Universal Robots PolyScope program: stopCollarMoveBottle.urp

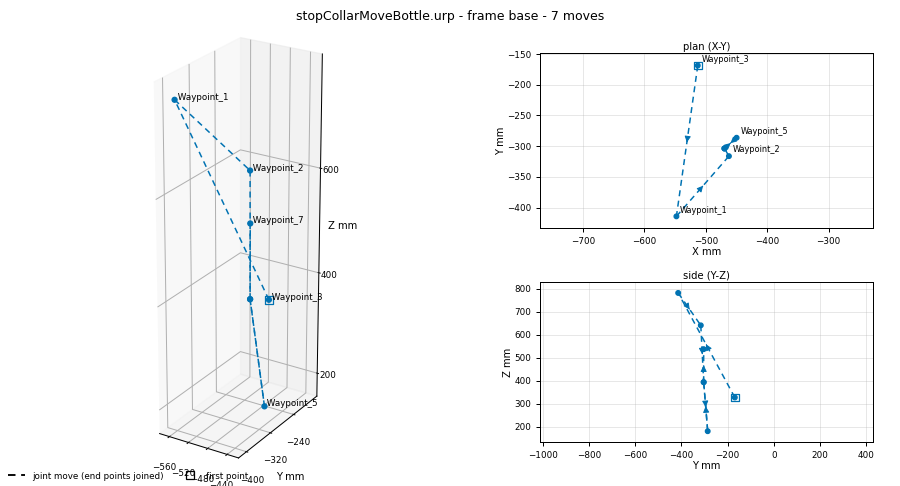
[picture p0: tool path of stopCollarMoveBottle.urp in frame base, 7 of 7 moves have a stored position in this frame; points joined in program order, loops and branches not executed]
Program stopCollarMoveBottle (installation=default directory=/programs/PrakjoyShi_Beer createdIn=5.12.6.1102099 lastSavedIn=5.12.6.1102099 robotSerialNumber=20215500597)
Calibrated DH parameters: a=[0.000193, -0.066673, -0.391568, -0.000012, 0.00005, 0]; d=[0.162643, -472.05677, 465.132521, 7.058239, 0.099746, 0.099582]; alpha=[1.571116, 0.00089, 0.003862, 1.569269, -1.569248, 0]; deltaTheta=[0, -1.413394, 7.628392, 0.068187, 0, -0.000001]
Robot Program (runOnlyOnce=true)
  MoveJ speed 60 deg/s, acceleration 80 deg/s^2 (useActiveTCP=true) feature=Base
    Waypoint Waypoint_3: TCP in base x=-512.964 y=-168.718 z=327.54 mm, rx=2.1022 ry=2.3346 rz=-0.0001 rad; joints [3.858, -85.637, 80.892, -85.168, -89.81, -2.096] deg; TCP offset x=0 y=0 z=191.5 mm, rx=0 ry=0 rz=0 rad
    URCap Gripper Activate (Robotiq_Grippers, Robotiq Inc.) dataModel(ResetAndActivateKey=false)
    Waypoint Waypoint_1: TCP in base x=-547.743 y=-414.347 z=780.951 mm, rx=1.0761 ry=1.4184 rz=-1.4361 rad; joints [-1.099, -77.445, 50.816, -80.12, -0.057, -0.124] deg
    Waypoint Waypoint_2: TCP in base x=-462.247 y=-316.309 z=640.386 mm, rx=-0.9397 ry=-1.5371 rz=1.7089 rad; joints [6.917, -110.667, 115.927, -188.919, -64.828, 6.848] deg
    Waypoint Waypoint_4: TCP in base x=-469.42 y=-303.764 z=393.89 mm, rx=-0.9663 ry=-1.499 rz=1.6747 rad; joints [6.93, -89.795, 142.192, -236.128, -67.835, 6.515] deg
    Waypoint Waypoint_5: TCP in base x=-449.734 y=-286.33 z=181.236 mm, rx=-0.8887 ry=-1.6496 rz=1.5115 rad; joints [1.734, -48.424, 150.987, -278.873, -61.761, -4.885] deg
    URCap Gripper (Robotiq_Grippers, Robotiq Inc.) dataModel(position=100.0, force=100.0, speed=100.0, positionInDouble=100.0, forceInDouble=100.0, speedInDouble=100.0, slaveIds=[9], blocking=true)
    Waypoint Waypoint_6: TCP in base x=-469.428 y=-303.765 z=393.886 mm, rx=-0.9663 ry=-1.499 rz=1.6747 rad; joints [6.929, -89.795, 142.191, -236.126, -67.832, 6.517] deg; TCP offset x=0 y=0 z=191.5 mm, rx=0 ry=0 rz=0 rad
    Waypoint Waypoint_7: TCP in base x=-469.423 y=-303.772 z=537.056 mm, rx=-0.9663 ry=-1.499 rz=1.6747 rad; joints [6.906, -106.663, 129.096, -206.192, -67.735, 6.591] deg; TCP offset x=0 y=0 z=191.5 mm, rx=0 ry=0 rz=0 rad
